FUNCTION_BLOCK FutureMCMoveAbsoluteCreator IMPLEMENTS InterfaceTaskCreator
VAR_INPUT
END_VAR
VAR_OUTPUT
END_VAR
VAR
	_axis: REFERENCE TO AXIS_REF;
	_position : MC_LREAL;
	_velocity : MC_LREAL;
	_acceleration: MC_LREAL;
	_deceleration: MC_LREAL;
	_jerk		: MC_LREAL;
	_option : ST_MoveOptions;
	_buffer_mode : MC_BufferMode ;
END_VAR

{warning 'add method implementation '}
METHOD create_future : InterfaceFuture
VAR_INPUT
	(* Specify future name*)
	future_name	: STRING;
END_VAR
VAR
	_p_future : POINTER TO FutureMCMoveAbsolute;
END_VAR
_p_future := __NEW(FutureMCMoveAbsolute);
_p_future^.future_name := future_name;
_p_future^.set_parameters(_axis, _position, _velocity, _acceleration, _deceleration,_jerk ,_buffer_mode);
_p_future^.set_options( _option);
create_future := _p_future^;
END_METHOD

{warning 'add method implementation '}
METHOD destroy_future : InterfaceFuture
VAR_INPUT
	(* Specify future instance whtat you want to delete.*)
	future	: InterfaceFuture;
END_VAR
VAR
	_p_future : POINTER TO FutureMCMoveAbsolute;
END_VAR
IF __QUERYPOINTER(future, _p_future) THEN
	__DELETE(_p_future);
	IF _p_future = 0  THEN
		destroy_future := 0;
	END_IF
END_IF
END_METHOD

METHOD set_options : BOOL
VAR_INPUT
	option : ST_MoveOptions;
END_VAR
_option := option;
END_METHOD

METHOD set_parameters : BOOL
VAR_INPUT
	axis : REFERENCE TO AXIS_REF;
	position : MC_LREAL;
	velocity : MC_LREAL;
	acceleration	: MC_LREAL;		// Set deceleration in case let moving axis halt.
	deceleration	: MC_LREAL;		// Set deceleration in case let moving axis halt.
	jerk			: MC_LREAL;		// Set jerk in case let moving axis halt.
	buffer_mode : MC_BufferMode;
END_VAR
_axis REF= axis;
_position := position;
_velocity := velocity;
_acceleration := acceleration;
_deceleration := deceleration;
_jerk := jerk;
_buffer_mode := buffer_mode;
END_METHOD

END_FUNCTION_BLOCK

(* stored: Version 1.1.0.1, ProductVersion 3.1.4024.15
   POU FutureMCMoveAbsoluteCreator: Id {c6c4289a-7217-4966-b462-57230d558786}, SpecialFunc None
   Method create_future: Id {21eef5d1-2501-4f7c-b086-fb969f968594}
   Method destroy_future: Id {5f5eec34-2256-4715-b6f4-85c5429d303d}
   Method set_options: Id {b3325934-92d7-4a4d-9778-7498306961eb}
   Method set_parameters: Id {0711e1be-0936-4a4c-bacb-b6283fd324ab} *)
